// Mitsubishi GX Works2 project: HMI 화면 전환, 언어 전환 코드   PLC: Q03UDV

PROGRAM MAIN
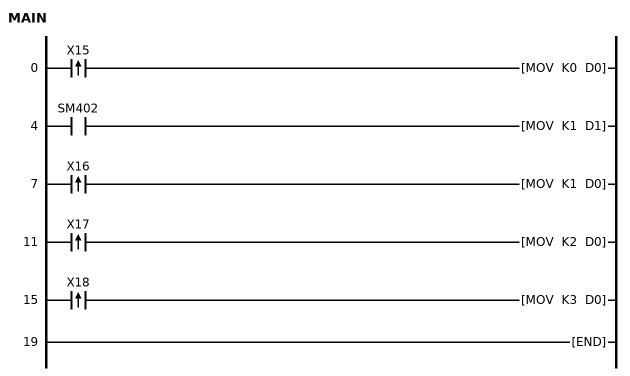
0     LDP     X15
      MOV     K0 D0
4     LD      SM402
      MOV     K1 D1
7     LDP     X16
      MOV     K1 D0
11    LDP     X17
      MOV     K2 D0
15    LDP     X18
      MOV     K3 D0
19    END
END_PROGRAM
